% RSLogix 500 project Rotameter.RSS, saved by version 8.30.00.16 %
PROJECT "UNTITLED"    % processor: Bul.1763 MicroLogix 1100 Series B %

PROGRAM FILES
  LAD 2   6 rungs

DATA FILES
  O0 OUTPUT  4 elements
  I1 INPUT  6 elements
  S2 STATUS  66 elements
  B3 BINARY  1 elements
  T4 TIMER  2 elements
  C5 COUNTER  1 elements
  R6 CONTROL  1 elements
  N7 INTEGER  1 elements
  F8 FLOAT  1 elements

LADDER 2
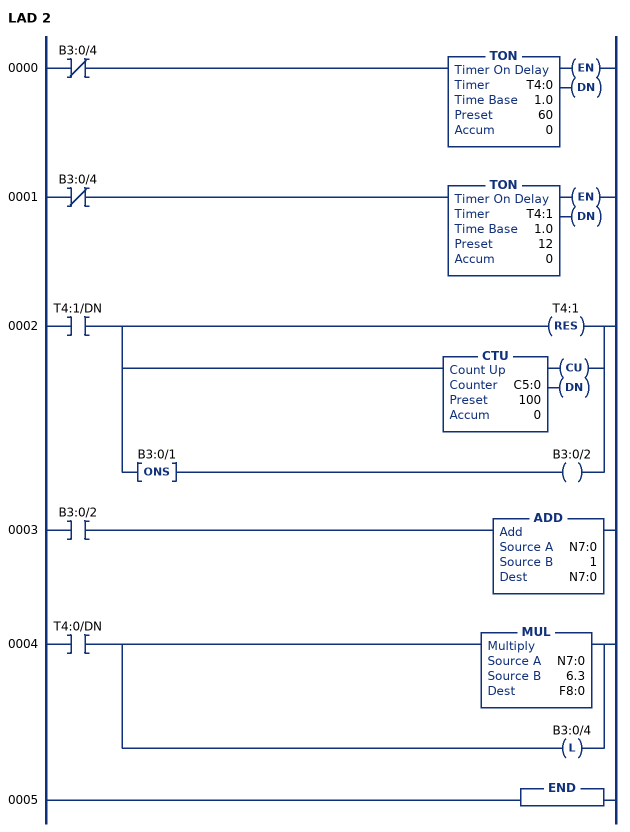
% Rung: 0 %
SOR XIO B3:0/4 TON T4:0 1.0 60 0 EOR
% Rung: 1 %
SOR XIO B3:0/4 TON T4:1 1.0 12 0 EOR
% Rung: 2 %
SOR XIC T4:1/DN BST RES T4:1 NXB CTU C5:0 100 0 NXB ONS B3:0/1 OTE B3:0/2 BND EOR
% Rung: 3 %
SOR XIC B3:0/2 ADD N7:0 1 N7:0 EOR
% Rung: 4 %
SOR XIC T4:0/DN BST MUL N7:0 6.3 F8:0 NXB OTL B3:0/4 BND EOR
% Rung: 5 %
SOR END EOR

DATA TABLE (non-zero values as saved)
DATA T4
% .PRE .ACC %
% T4:0 % 60 0
% T4:1 % 12 0
DATA C5
% .PRE .ACC %
% C5:0 % 100 0
